TYPE MachiningStation_DiscreteInputs :
STRUCT;
	EStop_Status		: BOOL;
	Door_State			: BOOL;
	Chuck_State			: BOOL;
	Stock_Present		: BOOL;
	Inspection_Pass		: BOOL;
	Inspection_Fail		: BOOL;
END_STRUCT
END_TYPE

(* stored: Version 1.1.0.1, ProductVersion 3.1.0.36
   DUT MachiningStation_DiscreteInputs: Id {8d55a58e-86d0-4190-ae66-aa67df72087b} *)
